DATA_BLOCK "ST10_StopperCtrl_DB"
{ S7_Optimized_Access := 'FALSE' }
VERSION : 0.1
NON_RETAIN
"ST10_StopperCtrl"

BEGIN

END_DATA_BLOCK

